{attribute 'GeneratedUsingTerminal: EL6001-0000-0020'}
{attribute addProperty BoxType "EL6001-0000-0020"}
{attribute addProperty Id "CtrlAT %Q*USINT1Data_OutAT %Q*ARRAY[0..2] OF USINT3"}
{attribute addProperty CRC "622567651"}
{attribute addProperty Size "4"}
TYPE Outputs_1EA34405 :
STRUCT
	{attribute addProperty Name "Ctrl"}
	Ctrl AT %Q* : USINT;
	{attribute addProperty Name "Data_Out"}
	Data_Out AT %Q* : ARRAY[0..2] OF USINT;
END_STRUCT
END_TYPE

(* stored: Version 1.2.0.0, ProductVersion 3.1.4024.9
   DUT Outputs_1EA34405: Id {0c1cf5e8-3bb3-4d7e-afca-2ab18ebb303e} *)
